// TIA Portal V20 export
TYPE "typeFeedbackFault"
// stored: Access Published, IsFailsafeCompliant true, Namespace Safety
   STRUCT
      MCFeedbackFault1 : Bool;   // Manifold1 Control Power FeedBack Fault
      MCFeedbackFault2 : Bool;   // FFU1 Control Power FeedBack Fault
      MCFeedbackFault3 : Bool;   // FFU2 Control Power FeedBack Fault
   END_STRUCT;
END_TYPE
